{attribute addProperty BoxType "EK1100-0000-0018"}
{attribute addProperty Id "Beckhoff_EL3xxx_0030EK1122Beckhoff_EL3xxx_0030EK1122_A8C7E601162A_0001_EL3174_0030_0016EL3174_83515A0D22428A_0002_EL3314_0030_0021EL3314_645580BD28836A_0003_EL3681_0030_0021EL3681_01269A6017622A_0004_EL3201_0030_0022EL3201_D2AFA85617722.125A_0005_EL3202_0030_0022EL3202_5359D6C325832.25A_0006_EL3356_0030_0025EL3356_CA56400F16020A_0007_EL3692_0030_0021EL3692_3E4349A528836"}
{attribute addProperty CRC "3287359125"}
{attribute addProperty SizeInBites "1587"}
{attribute addProperty SizeInBytes "198.375"}
TYPE Beckhoff_EL3xxx_0030_C3F11E95 EXTENDS EK1100_179A0949 :
STRUCT
	{attribute addProperty Name "Beckhoff_EL3xxx_0030EK1122"}
	Beckhoff_EL3xxx_0030EK1122 : Beckhoff_EL3xxx_0030EK1122_A8C7E601;
	{attribute addProperty Name "A_0001_EL3174_0030_0016"}
	A_0001_EL3174_0030_0016 : EL3174_83515A0D;
	{attribute addProperty Name "A_0002_EL3314_0030_0021"}
	A_0002_EL3314_0030_0021 : EL3314_645580BD;
	{attribute addProperty Name "A_0003_EL3681_0030_0021"}
	A_0003_EL3681_0030_0021 : EL3681_01269A60;
	{attribute addProperty Name "A_0004_EL3201_0030_0022"}
	A_0004_EL3201_0030_0022 : EL3201_D2AFA856;
	{attribute addProperty Name "A_0005_EL3202_0030_0022"}
	A_0005_EL3202_0030_0022 : EL3202_5359D6C3;
	{attribute addProperty Name "A_0006_EL3356_0030_0025"}
	A_0006_EL3356_0030_0025 : EL3356_CA56400F;
	{attribute addProperty Name "A_0007_EL3692_0030_0021"}
	A_0007_EL3692_0030_0021 : EL3692_3E4349A5;
END_STRUCT
END_TYPE

(* stored: Version 1.2.0.0, ProductVersion 3.1.4024.9
   DUT Beckhoff_EL3xxx_0030_C3F11E95: Id {783b6d4e-d3e1-492a-8134-4cfb2579c5d8} *)
